Universal Robots URScript: step1_full_no_contact_pipeline.script

# Step1: full no-contact pipeline dry run.
# This is the final contact-run scaffold without contact search or force
# control. It requires the Python Kunwei RTDE bridge to be running.
#
# Boundary:
# - fixed TCP orientation unless use_reference_orientation is set to 1
# - move to reference XY start at current Z, never to the old contact Z
# - software zero request only, no UR zero_ftsensor and no Kunwei tare
# - no z-down search and no normal-force correction

def codex_abs(x):
  if x < 0.0:
    return -x
  end
  return x
end

def codex_wait_for_sensor_ok(timeout_s):
  local dt = 0.008
  local t = 0.0
  while t < timeout_s:
    if read_input_float_register(27) > 0.5:
      return True
    end
    sync()
    t = t + dt
  end
  return False
end

def codex_guard_ok():
  local normal_force = read_input_float_register(24)
  local force_norm = read_input_float_register(25)
  local sensor_ok = read_input_float_register(27)
  local stop_request = read_input_float_register(28)
  local torque_norm = read_input_float_register(30)
  if sensor_ok < 0.5:
    return False
  elif stop_request > 0.5:
    return False
  elif codex_abs(normal_force) > 12.0:
    return False
  elif force_norm > 15.0:
    return False
  elif torque_norm > 0.6:
    return False
  end
  return True
end

def codex_step1_full_no_contact_pipeline():
  local ux = 0.679764156
  local uy = -0.733430768
  local path_start_x = 0.446585764
  local path_start_y = 0.226717001
  local ref_rx = 3.141572714
  local ref_ry = -0.000026465
  local ref_rz = -0.000024158
  local use_reference_orientation = 0
  local approach_speed_m_s = 0.010
  local tangent_speed_m_s = 0.005
  local path_length_m = 0.06358
  local path_progress_min_m = -0.003
  local path_progress_max_m = 0.067
  local path_runtime_limit_s = 18.0
  local retract_z_m = 0.050
  local retract_speed_m_s = 0.005
  local dt = 0.008
  local stop_reason = 0.0

  textmsg("codex step1 full no-contact pipeline start")

  # 0. Sensor stream and initial software zero must already be good.
  write_output_float_register(35, 0.0)
  if not codex_wait_for_sensor_ok(3.0):
    stop_reason = 3.0
  end

  # 1. Move to target path start XY at current Z. Orientation correction is
  # intentionally gated by use_reference_orientation.
  if stop_reason == 0.0:
    write_output_float_register(35, 1.0)
    local p0 = get_actual_tcp_pose()
    local target_start = p[path_start_x, path_start_y, p0[2], p0[3], p0[4], p0[5]]
    if use_reference_orientation > 0.5:
      target_start = p[path_start_x, path_start_y, p0[2], ref_rx, ref_ry, ref_rz]
    end
    movel(target_start, a=0.030, v=approach_speed_m_s, r=0.0)
    stopl(0.5)
  end

  # 2. Request a second software ftzero at the path start.
  if stop_reason == 0.0:
    write_output_float_register(35, 2.0)
    local zero_request = read_input_float_register(26)
    write_output_float_register(34, zero_request)
    sleep(0.20)
    if not codex_wait_for_sensor_ok(3.0):
      stop_reason = 3.0
    end
  end

  # 3. Guard is active before and during the no-contact XY motion.
  if stop_reason == 0.0 and not codex_guard_ok():
    stop_reason = 4.0
  end

  # 4. Contact search placeholder: skipped for Step1.
  if stop_reason == 0.0:
    write_output_float_register(35, 4.0)
  end

  # 5. Force-control placeholder: skipped for Step1.
  if stop_reason == 0.0:
    write_output_float_register(35, 5.0)
  end

  # 5.1. Execute the full XY dry-run line at fixed Z.
  if stop_reason == 0.0:
    write_output_float_register(35, 5.1)
    local start_pose = get_actual_tcp_pose()
    local t = 0.0
    while stop_reason == 0.0:
      local pose_now = get_actual_tcp_pose()
      local dx = pose_now[0] - start_pose[0]
      local dy = pose_now[1] - start_pose[1]
      local progress_m = dx * ux + dy * uy
      write_output_float_register(30, stop_reason)
      write_output_float_register(31, progress_m)
      write_output_float_register(32, 0.0)
      write_output_float_register(33, 0.0)
      if not codex_guard_ok():
        stop_reason = 4.0
      elif progress_m >= path_length_m:
        stop_reason = 1.0
      elif progress_m < path_progress_min_m or progress_m > path_progress_max_m:
        stop_reason = 9.0
      elif t > path_runtime_limit_s:
        stop_reason = 10.0
      else:
        speedl([ux * tangent_speed_m_s, uy * tangent_speed_m_s, 0.0, 0.0, 0.0, 0.0], 0.03, dt)
        sync()
        t = t + dt
      end
    end
    stopl(0.5)
  end

  # 6. Retract: keep XY unchanged, move +Z.
  if stop_reason == 1.0:
    write_output_float_register(35, 6.0)
    local retract_start = get_actual_tcp_pose()
    local retract_done = False
    while not retract_done:
      local pose_now = get_actual_tcp_pose()
      local dz = pose_now[2] - retract_start[2]
      write_output_float_register(32, dz)
      if dz >= retract_z_m:
        retract_done = True
      else:
        speedl([0.0, 0.0, retract_speed_m_s, 0.0, 0.0, 0.0], 0.03, dt)
        sync()
      end
    end
    stopl(0.5)
  end

  write_output_float_register(30, stop_reason)
  textmsg("codex step1 full no-contact pipeline stop reason:", stop_reason)
end

codex_step1_full_no_contact_pipeline()
